TYPE STMStatus :
STRUCT
	readyToEnable : BOOL;
	ready : BOOL;
	warning : BOOL;
	error : BOOL;
	movingPositive : BOOL;
	movingNegative : BOOL;
	txPDOToggle : BOOL;
END_STRUCT
END_TYPE

(* stored: Version 1.1.0.1, ProductVersion 3.1.4024.11
   DUT STMStatus: Id {b5bb59d1-b29b-4e4e-95c7-ce1c9592a19e} *)
